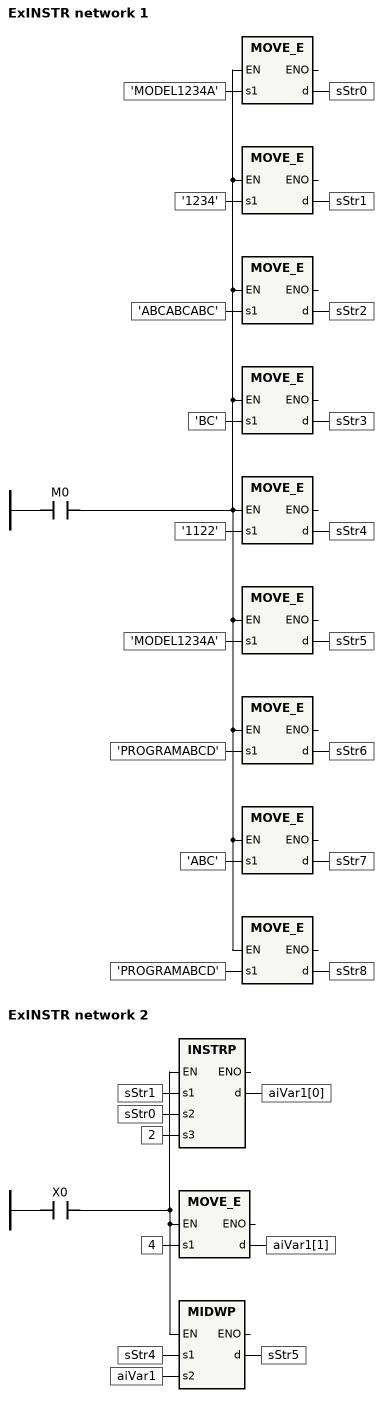
(* [picture p24: structured ladder/FBD of ExINSTR, networks 1 to 2] *)
(* network 1 *)
MOVE_E(M0, 'MODEL1234A', sStr0);
MOVE_E(M0, '1234', sStr1);
MOVE_E(M0, 'ABCABCABC', sStr2);
MOVE_E(M0, 'BC', sStr3);
MOVE_E(M0, '1122', sStr4);
MOVE_E(M0, 'MODEL1234A', sStr5);
MOVE_E(M0, 'PROGRAMABCD', sStr6);
MOVE_E(M0, 'ABC', sStr7);
MOVE_E(M0, 'PROGRAMABCD', sStr8);
(* network 2 *)
INSTRP(X0, sStr1, sStr0, 2, aiVar1[0]);
MOVE_E(X0, 4, aiVar1[1]);
MIDWP(X0, sStr4, aiVar1, sStr5);
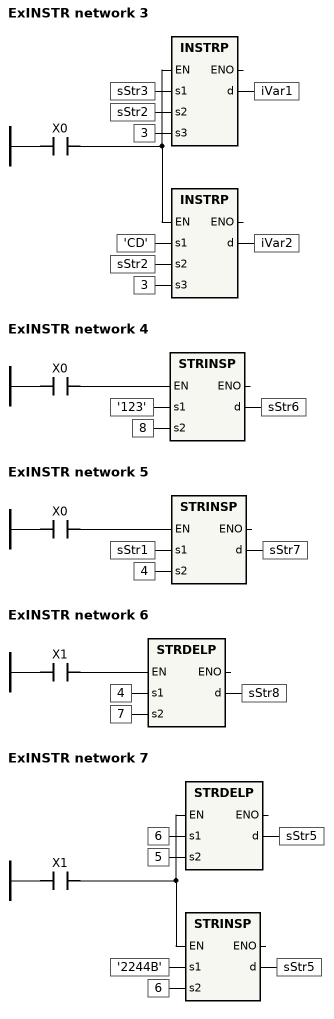
(* network 3 *)
INSTRP(X0, sStr3, sStr2, 3, iVar1);
INSTRP(X0, 'CD', sStr2, 3, iVar2);
(* network 4 *)
STRINSP(X0, '123', 8, sStr6);
(* network 5 *)
STRINSP(X0, sStr1, 4, sStr7);
(* network 6 *)
STRDELP(X1, 4, 7, sStr8);
(* network 7 *)
STRDELP(X1, 6, 5, sStr5);
STRINSP(X1, '2244B', 6, sStr5);
END_PROGRAM
